// TwinCAT 3 PLC project AxisIaiLib
// Title: AxisIaiLibrary
// Company: Gema
// Author: RG
// ProjectVersion: 0.0.0.1
// ProgramVersion: 3.1.4024.0
// libraries:
//   Tc2_Standard, * (Beckhoff Automation GmbH)
//   TcoCore, 0.11.0.35 (Vortex.Library)
//   TcoData, 0.11.0.35 (Vortex.Library)
//   TcoDrivesBeckhoff, 0.11.0.35 (Vortex.Library)
//   TcoElements, 0.11.0.35 (Vortex.Library)
//   TcoIo, 0.11.0.35 (Vortex.Library)
//   TcoPneumatics, 0.11.0.35 (Vortex.Library)
//   TcoUtilities, 0.11.0.35 (Vortex.Library)
// project tree:
//   Context/ MainStation.TcPOU (not stored), PRG_TEST.TcPOU, TcUnitContext.TcPOU
//   IAI/Data types/ AxisLimits.TcDUT (not stored), IAIAxisStatus.TcDUT (not stored), IOAxis.TcDUT
//   IAI/Data types/Enum/ eSetPositionMode.TcDUT, E_AccelMode.TcDUT (not stored), E_RMod.TcDUT (not stored), E_StopMode.TcDUT (not stored)
//   IAI/Data types/Interfaces/ iSuperActuator.TcIO
//   IAI/Data types/In/Gateway/ GatewayStatus.TcDUT, StatusSignal0.TcDUT, StatusSignal1.TcDUT
//   IAI/Data types/In/ PlcIn.TcDUT, StatusIn.TcDUT
//   IAI/Data types/Out/ ControlOut.TcDUT, PlcOut.TcDUT
//   IAI/Data types/Out/Gateway/ ControlSignal0.TcDUT, ControlSignal1.TcDUT, GatewayControl.TcDUT (not stored)
//   IAI/Global Variables/ AxisStats.TcGVL, AxisStatsGlobal.TcGVL
//   IAI/IAI_Drive/TcoAxis/ AxisIAI.TcPOU, IAxisIAI.TcIO, Power.TcPOU
//   IAI/IAI_Drive/TcoAxis/AxisTasks/ ResetTask.TcPOU, SetPositionTask.TcPOU
//   IAI/IAI_Drive/TcoAxis/MotionTasks/ HaltTask.TcPOU, HomeTask.TcPOU, MoveAbsoluteTask.TcPOU, MoveRelativeTask.TcPOU, StopTask.TcPOU
// (motion and I/O tree: see PLC project axisiailibexample)
// real-time tasks:
//   TASK PlcTask: cycle T#10ms, priority 20, ADS port 350

// ---- IAI/Data types/Enum/eSetPositionMode.TcDUT
{attribute 'qualified_only'}
{attribute 'strict'}
TYPE
    eSetPositionMode :
    (
        Absolute := 0,
        Relative := 1
    );
END_TYPE

// ---- IAI/Data types/In/Gateway/GatewayStatus.TcDUT
TYPE
    GatewayStatus :
    STRUCT
        GatewayStatus0 : StatusSignal0;
        GatewayStatus1 : StatusSignal1;
        AnswerCmd      : WORD;
        Data0          : WORD;
        Data1          : WORD;
        Data2          : WORD;
        Data3          : WORD;
        UsedSpace      : WORD;
    END_STRUCT
END_TYPE

// ---- IAI/Data types/In/Gateway/StatusSignal0.TcDUT
TYPE
    StatusSignal0 :
    STRUCT
        //~
        ALMC1 : USINT; //Alarmcode from Gateway
        SEMG  : BIT;   //EMGIN off, --> Emergency Stop
        b9    : BIT;
        ALML  : BIT; // easy Error in Gateway, wrong Paramter
        ALMH  : BIT; // Sever Error in Gaateway, wrong Parameter, Rerstart req
        MODE  : BIT; // True if Mode = Manu
        ERRT  : BIT; //COMM Err between Axis and Gaetway
        LERC  : BIT; //ERror while Run  ERR-T or ERR-C in Gateway
        RUN   : BIT; //Running Gateway
    //~
    END_STRUCT
END_TYPE

// ---- IAI/Data types/In/Gateway/StatusSignal1.TcDUT
TYPE
    StatusSignal1 :
    STRUCT
        //~
        LNK0 : BIT; // zeigt aktive Achsennummer im Gateway
        LNK1 : BIT; // zeigt aktive Achsennummer im Gateway
        LNK2 : BIT; // zeigt aktive Achsennummer im Gateway
        LNK3 : BIT; // zeigt aktive Achsennummer im Gateway
        LNK4 : BIT; // zeigt aktive Achsennummer im Gateway
        LNK5 : BIT; // zeigt aktive Achsennummer im Gateway
        LNK6 : BIT; // zeigt aktive Achsennummer im Gateway
        LNK7 : BIT; // zeigt aktive Achsennummer im Gateway
        MNT0 : BIT; // Bit for Easy Error
        MNT1 : BIT; // Bit for Easy Error
        MNT2 : BIT; // Bit for Easy Error
        MNT3 : BIT; // Bit for Easy Error
        MNT4 : BIT; // Bit for Easy Error
        MNT5 : BIT; // Bit for Easy Error
        MNT6 : BIT; // Bit for Easy Error
        MNT7 : BIT; // Bit for Easy Error
    //~
    END_STRUCT
END_TYPE

// ---- IAI/Data types/In/PlcIn.TcDUT
TYPE
    PlcIn :
    //    (*PCON-CA output -> PLC input  - 32 bytes *)
    STRUCT
        CurrentPosition : DINT; (*Unit: 0,01mm*)
        CommandCurrent  : DINT; (*Unit: mA*)
        CurrentSpeed    : UINT; (*Unit: 0,01mm/s*)
        Unavailable1    : WORD; (*n+14;n+15*)
        AlarmCode       : UINT; (*0- no Error*)
        //        TotalMovingCount : UDINT; (*Unit: times*)
        //        TotalMovingDistance : UDINT; (*Unit: m*)
        StatusSignal : StatusIn;
    //        StatusSignal2 : WORD; (*n+30;n+31*)
    END_STRUCT
END_TYPE

// ---- IAI/Data types/In/StatusIn.TcDUT
TYPE
    StatusIn :
    STRUCT
        //~
        PEND  : BIT; //Signal wird true nach Abschluss Positionierung, on during Stop if Motor on
        HEND  : BIT; //True after Homeing, until Pos lost
        MOVE1 : BIT; //True while Moving
        ALM   : BIT; // true while Alarm
        SV    : BIT; //True when ready, (Servo On)
        PSFL  : BIT; //True while Error in SchubBetrieb
        bit6  : BIT;
        ALML  : BIT; //izi Error
        MEND  : BIT; //Signal True after Moving, Homing or Schubvorgang, False by Start new Movement
        bit9  : BIT;
        bit10 : BIT;
        bit11 : BIT;
        ZONE1 : BIT; // True when in Zone1
        ZONE2 : BIT;
        CRDY  : BIT; // Controller in Standby
        EMGS  : BIT; // Emergency Stop
    //~
    END_STRUCT
END_TYPE

// ---- IAI/Data types/IOAxis.TcDUT
TYPE
    IOAxis :
    STRUCT
        GateWayStatus  : GatewayStatus;
        GateWayControl : GatewayControl;
        PlcInFromAxis  : PlcIn;
        PlcOutToAxis   : PlcOut;
    END_STRUCT
END_TYPE

// ---- IAI/Data types/Out/ControlOut.TcDUT
TYPE
    ControlOut :
    STRUCT
        //~
        CSTR        : BIT; // Positionierungs Start, Trigger
        HOME        : BIT; // Referenzfahrt
        STP         : BIT; // PAuse
        RES         : BIT; // REset
        SON         : BIT; //Servo Ein
        JISL        : BIT; //Wechsel zwischen Jog/Inch Betrieb
        JVEL        : BIT; // Umschalten von Jog-Geschw/Schrittweite  S119 ANleitung
        JOGNegative : BIT; //-Jog
        JOGPositive : BIT; //+Jog
        b9          : BIT;
        b10         : BIT;
        b11         : BIT;
        PUSH        : BIT; //Schubbetrieb, True = Schubbetrieb, False = Positionierbetrieb
        DIR         : BIT; //Schubrichtung, True = Entgegen Refernezpunktrichtung
        INC         : BIT; //False= Absolute Positionsbefehle, True = Inkrementale
        BKRL        : BIT; //True = Bremsfreigabe, False = Bremse aktiv
    //~
    END_STRUCT
END_TYPE

// ---- IAI/Data types/Out/Gateway/ControlSignal0.TcDUT
TYPE
    ControlSignal0 :
    STRUCT
        //~
        b0  : BIT;
        b1  : BIT;
        b2  : BIT;
        b3  : BIT;
        b4  : BIT;
        b5  : BIT;
        b6  : BIT;
        b7  : BIT;
        b8  : BIT;
        b9  : BIT;
        b10 : BIT;
        b11 : BIT;
        b12 : BIT;
        RTE : BIT; //ERR-T oder ERR-C REset during Run
        b14 : BIT;
        MON : BIT; //must be on, Controll with Communication active
    //~
    END_STRUCT
END_TYPE

// ---- IAI/Data types/Out/Gateway/ControlSignal1.TcDUT
TYPE
    ControlSignal1 :
    STRUCT
        word1 : word;
    END_STRUCT
END_TYPE

// ---- IAI/Data types/Out/PlcOut.TcDUT
TYPE
    PlcOut :
    //    (*PCON-CA output -> PLC input  - 32 bytes *)
    STRUCT
        TargetPosition  : DINT := 1000; (*Unit: 0,01 mm*)
        PositioningBand : DINT := 10;   (*Unit: 0,01 mm or pressing width value*)
        Velocity        : UINT := 1;    (*Unit 0,01 mm/s*)
        //        ZoneBoundary_pos : DINT; (*Unit 0,01 mm*)
        //        ZoneBoundary_neg : DINT; (*Unit 0,01 mm*) (*pos >= neg!*)
        Accelerartion : UINT := 1; (*Acc und Dec Unit: 0,01 G*) (*Range 1.. 300*)
        //        Decelerartion : UINT; (*Unit: 0,01 G*) (*Range 1.. 300*)
        //        PressingCurrentLimitValue : UINT; (*Unit: %*) (*Range 0(0%) .. 510(200%)*)
        PushCurrentLimit : UINT := 1; (*Schubstrombegrenzung Unit: %*) (*Range 0(0%) .. 255(100%)*)
        ControlSignal    : ControlOut;                                 (*n+28;n+29*)
    //        ControlSignal2 : WORD; (*n+30;n+31*)
    END_STRUCT
END_TYPE

// ---- IAI/Global Variables/AxisStats.TcGVL
{attribute 'Tc2GvlVarNames'}
{attribute 'qualified_only'}
VAR_GLOBAL CONSTANT

    AxisLimitsRfid     : AxisLimits := (MaxAcceleration := 100, MaxPosition := 20000, MaxVelocity := 900);
    AxisLimitsAssembly : AxisLimits := (MaxAcceleration := 100, MaxPosition := 25000, MaxVelocity := 900);
    AxisLimitsMounting : AxisLimits := (MaxAcceleration := 100, MaxPosition := 40000, MaxVelocity := 840);

END_VAR

// ---- IAI/Global Variables/AxisStatsGlobal.TcGVL
{attribute 'Tc2GvlVarNames'}
{attribute 'qualified_only'}
VAR_GLOBAL CONSTANT
    MaxAcceleration1 : UINT := 100;
    MINPosition1     : DINT := 0;
    MaxPosition1     : DINT := 20000;
    MaxVelocity1     : UINT := 900;

    MaxAcceleration2 : UINT := 100;
    MINPosition2     : DINT := 0;
    MaxPosition2     : DINT := 25000;
    MaxVelocity2     : UINT := 900;

    MaxAcceleration3 : UINT := 100;
    MINPosition3     : DINT := 0;
    MaxPosition3     : DINT := 40000;
    MaxVelocity3     : UINT := 840;

END_VAR

// ---- IAI/Data types/Interfaces/iSuperActuator.TcIO
INTERFACE iSuperActuator

METHOD ErrorHandling : BOOL
VAR_INPUT
END_VAR
END_METHOD

PROPERTY IsError : bool
GET
END_GET
END_PROPERTY

METHOD ResetError : BOOL
VAR_INPUT
END_VAR
END_METHOD

END_INTERFACE

// ---- IAI/IAI_Drive/TcoAxis/IAxisIAI.TcIO
INTERFACE IAxisIAI

PROPERTY DriveRef : REFERENCE TO AxisIAI
GET
END_GET
END_PROPERTY

END_INTERFACE

// ---- Context/PRG_TEST.TcPOU
PROGRAM PRG_TEST
VAR
    _testSuite : TcUnitContext;
END_VAR

_testSuite.Run();
_testSuite.RtcSynchronize(true, '', 60);

END_PROGRAM

// ---- Context/TcUnitContext.TcPOU
FUNCTION_BLOCK TcUnitContext EXTENDS TcoCore.TcoContext
VAR
    _mainStation : MainStation(THIS^);

    {attribute addProperty Name "Versionsnummer Plc"}
    _sVersion : STRING(23);
    //~
    _stProgramVersion : ST_LibVersion;
    //~

END_VAR

(*~
    <docu>
        <summary>
            Main method of the TcoContext. This is the entry point of any control logic that belongs to this context.
            The call of this method is ensured by calling the <c>InstanceName.Run()</c> method, and it must not be called explicitly.
            This method is abstract, and it must be overridden in derived block.
        </summary>
    </docu>
~*)
METHOD PROTECTED Main

_mainStation();
END_METHOD

END_FUNCTION_BLOCK

// ---- IAI/IAI_Drive/TcoAxis/AxisIAI.TcPOU
FUNCTION_BLOCK AxisIAI EXTENDS TcoCore.TcoComponent IMPLEMENTS IAxisIAI, iSuperActuator
VAR_INPUT
    inEnabled : BOOL; // Power ein
END_VAR
VAR_OUTPUT
END_VAR
VAR_IN_OUT
    GateWayStatus  : GatewayStatus;
    GateWayControl : GatewayControl;

    DriveToPlc : PlcIn;
    PlcToDrive : PlcOut;

END_VAR
VAR
    //    _baseAxis : FB_SpecialControl(maxAcc := _maxAcc, minPos := _minPos, maxPos := _maxPos, maxVel := _maxVel);
    {attribute clr [ReadOnly()]}
    _axisStatus : IAIAxisStatus;
    _axisLimit  : AxisLimits;

    {attribute 'hide'}
    _sb        : TcoCore.StringBuilder;
    _errorDesc : string;
END_VAR
VAR
    _power : Power(THIS^);
    {attribute addProperty Name "Referenz (Aufpassen)"}
    _homeTask : HomeTask(THIS^);
    {attribute addProperty Name "<#Reset#>"}
    _resetTask : ResetTask(THIS^);
    {attribute addProperty Name "<#Set position#>"}
    _setPositionTask : SetPositionTask(THIS^);
    //	    {attribute addProperty Name "<#Jogging#>"}
    //    _jog : Jog(THIS^);
    {attribute addProperty Name "<#Stop#>"}
    _stopTask : StopTask(THIS^);
    {attribute addProperty Name "<#Halt#>"}
    _haltTask : HaltTask(THIS^);
    {attribute addProperty Name "<#Move relative#>"}
    _moveRelativeTask : MoveRelativeTask(THIS^);
    {attribute addProperty Name "<#Move absolute#>"}
    _moveAbsoluteTask : MoveAbsoluteTask(THIS^);
    //    {attribute addProperty Name "<#Move modulo#>"}
    //    _moveModuloTask : MoveModuloTask(THIS^);
    _faultTask : TcoCore.TcoTask(THIS^);
END_VAR


UpdateAxisStatus();

_power(inEnable := inEnabled);

_resetTask();

_homeTask();
_setPositionTask();
_stopTask();
_haltTask();
_moveRelativeTask();
_moveAbsoluteTask();
THIS^.Service();
//_moveModuloTask();

IF (_axisStatus.Error) THEN
    CASE _axisStatus.ErrorId OF
        111:
            _errorDesc := 'NotAus der Achse, bitte Checken';
        131:
            _errorDesc := 'Referenzfahrt nicht Complete';
        163:
            _errorDesc := 'Position Command Data invalid';
        193:
            _errorDesc := '0C1,Fehler Achse, Motorlast zu hoch aufgrund externer Kraft';
        333, 444, 555:
            _errorDesc := 'Servo ist aus';

    ELSE
        _errorDesc := 'For details see the service mode';

    END_CASE

    Messenger.Error
    (
        _sb.Clear()
            .Append('<#Drive error no #>')
            .Append(UDINT_TO_STRING(_axisStatus.ErrorId))
            .Append(': ')
            .Append(_errorDesc)
            .ToString()
    );

    _faultTask.ThrowWhen(TRUE);
END_IF;

UpdateAxisStatus();

PROPERTY AxisStatus : REFERENCE TO IAIAxisStatus
GET
UpdateAxisStatus();
AxisStatus REF= _axisStatus;
END_GET
END_PROPERTY

METHOD INTERNAL ClearError
_axisStatus.Error   := FALSE;
_axisStatus.ErrorId := 0;
END_METHOD

PROPERTY DriveRef : REFERENCE TO AxisIAI
GET
IF __ISVALIDREF(DriveRef) THEN
    DriveRef := THIS^;
end_if
END_GET
END_PROPERTY

METHOD ErrorHandling : BOOL
END_METHOD

PROPERTY FaultTask : TcoCore.ITcoTask
GET
FaultTask := _faultTask;
END_GET
END_PROPERTY

{attribute 'hide'}
METHOD FB_init : BOOL
VAR_INPUT
    bInitRetains : BOOL; // if TRUE, the retain variables are initialized (warm start / cold start)
    bInCopyCode  : BOOL; // if TRUE, the instance afterwards gets moved into the copy code (online change)
    ParentObject : ITcoObject;
    AxisLimits   : AxisLimits;
END_VAR
SUPER^.FB_init(bInitRetains, bInCopyCode, ParentObject);

THIS^._axisLimit := AxisLimits;
END_METHOD

METHOD Halt : ITcoTaskStatus
VAR_INPUT
    inDeceleration : UINT;
END_VAR
Halt := THIS^._haltTask.InvokeWithParams(inDeceleration := inDeceleration);
END_METHOD

PROPERTY HaltTask : TcoCore.ITcoTaskStatus
GET
HaltTask := _haltTask;
END_GET
END_PROPERTY

PROPERTY HomeTask : TcoCore.ITcoTaskStatus
GET
HomeTask := _homeTask;
END_GET
END_PROPERTY

PROPERTY isEnabled : BOOL
GET
isEnabled := inEnabled and DriveToPlc.StatusSignal.SV;
END_GET
END_PROPERTY

PROPERTY IsError : BOOL
GET
IsError := _faultTask.Error;
END_GET
END_PROPERTY

METHOD MoveAbsolute : ITcoTaskStatus
VAR_INPUT
    TargetPosition   : REAL;
    PositionBand     : REAL;
    Velocity         : UINT;
    Acceleration     : UINT;
    PushCurrentLimit : USINT;
END_VAR
MoveAbsolute := THIS^._moveAbsoluteTask.InvokeWithParams
(
    TargetPosition     := TargetPosition
    , PositionBand     := PositionBand
    , Velocity         := Velocity
    , Acceleration     := Acceleration
    , PushCurrentLimit := PushCurrentLimit
);
END_METHOD

PROPERTY MoveAbsoluteTask : TcoCore.ITcoTaskStatus
GET
MoveAbsoluteTask := _moveAbsoluteTask;
END_GET
END_PROPERTY

METHOD MoveHome : ITcoTaskStatus
VAR_INPUT
END_VAR
MoveHome := _homeTask.Invoke();
END_METHOD

METHOD MoveRelative : ITcoTaskStatus
VAR_INPUT
    Distance         : REAL;
    PositionBand     : REAL;
    Velocity         : UINT;
    Acceleration     : UINT;
    PushCurrentLimit : USINT;
END_VAR
MoveRelative := THIS^._moveRelativeTask.InvokeWithParams
(
    Distance           := Distance
    , Velocity         := Velocity
    , Acceleration     := Acceleration
    , PositionBand     := PositionBand
    , PushCurrentLimit := PushCurrentLimit
);
END_METHOD

PROPERTY MoveRelativeTask : TcoCore.ITcoTaskStatus
GET
MoveRelativeTask := _moveRelativeTask;
END_GET
END_PROPERTY

METHOD Reset : ITcoTaskStatus
Reset := THIS^._resetTask.Invoke();
ClearError();
END_METHOD

METHOD ResetError : BOOL
Restore();
END_METHOD

PROPERTY ResetTask : TcoCore.ITcoTaskStatus
GET
ResetTask := _resetTask;
END_GET
END_PROPERTY

(*~
    <docu>
        <summary>
            Restores this instance to the Ready state. Can be called explicitly or from within one of the restore mechanisms.
        </summary>
    </docu>
~*)
METHOD Restore : ITcoRestorable
Reset();
RestoreTasks();
END_METHOD

METHOD RestoreTasks : ITcoRestorable
VAR_INPUT
END_VAR
//Restore all
_homeTask.Restore();
_resetTask.Restore();
_setPositionTask.Restore();
_stopTask.Restore();
_haltTask.Restore();
_moveRelativeTask.Restore();
_moveAbsoluteTask.Restore();
_resetTask.Restore();
_faultTask.Restore();
END_METHOD

(*~
    <docu>
        <summary>
            Custom service (manual, maintenance) logic.
            This method must be implemented in derived class.
        </summary>
    </docu>
~*)
METHOD PROTECTED ServiceMode
//_jog.Service();
END_METHOD

METHOD INTERNAL SetErrorID
VAR_INPUT
    inErrorId : UDINT;
END_VAR
_axisStatus.Error := TRUE;

IF inErrorId <> 0 THEN
    _axisStatus.ErrorId := inErrorId;
ELSIF DriveToPlc.StatusSignal.EMGS THEN
    _axisStatus.ErrorId := 111;
END_IF
END_METHOD

METHOD SetPosition : ITcoTaskStatus
VAR_INPUT
    inPosition : LREAL;
    inMode     : eSetPositionMode;
END_VAR
SetPosition := THIS^._setPositionTask.InvokeWithParams(inPosition := inPosition, inMode := inMode);
END_METHOD

PROPERTY SetPositionTask : TcoCore.ITcoTaskStatus
GET
SetPositionTask := _setPositionTask;
END_GET
END_PROPERTY

METHOD Stop : ITcoTaskStatus
VAR_INPUT
    inDeceleration : UINT;
END_VAR
Stop := THIS^._stopTask.InvokeWithParams(inDeceleration := inDeceleration);
END_METHOD

PROPERTY StopTask : TcoCore.ITcoTaskStatus
GET
StopTask := _stopTask;
END_GET
END_PROPERTY

METHOD INTERNAL UpdateAxisStatus
VAR
    _message : STRING(125);
END_VAR
_axisStatus.ActPos := DriveToPLC.CurrentPosition / 100.0;
//_axisStatus.ModuloActPos := AxisRef.NcToPlc.ModuloActPos;
//_axisStatus.ModuloActTurns := AxisRef.NcToPlc.ModuloActTurns;
_axisStatus.ActVelo := DriveToPLC.CurrentSpeed;
//_axisStatus.ActAcc := AxisRef.NcToPlc.ActAcc;
_axisStatus.ActTorque := DriveToPLC.CommandCurrent;
//_axisStatus.CmdNo := AxisRef.NcToPlc.CmdNo;
//_axisStatus.CmdState := AxisRef.NcToPlc.CmdState;

//IF NOT Tc2MC2_TO_Tco_AxisStates(AxisRef.Status.MotionState, _axisStatus.MotionState) THEN
//    _message := Tc2_Standard
//        .CONCAT('Unable to cast AxisRef.Status.MotionState variable of type Tc2_MC2.MC_AxisStates (', TO_STRING(AxisRef.Status.MotionState));

//    _message := Tc2_Standard.CONCAT(_message, ') to the type TcoDrivesBeckhoff.eAxisStates!!!');
//    THIS^.Messenger.Post(_message, TcoCore.eMessageCategory.ProgrammingError);
//END_IF

//AlarmCodes ausprogrammieren (alle Gateway ALarmcodes etc.)
IF (DriveToPLC.StatusSignal.ALM OR DriveToPLC.StatusSignal.ALML or DriveToPlc.StatusSignal.EMGS) THEN
    SetErrorID(DriveToPlc.AlarmCode);
END_IF

//_axisStatus.ErrorStop := AxisRef.Status.ErrorStop;
//_axisStatus.Disabled := AxisRef.Status.Disabled;
//_axisStatus.Stopping := AxisRef.Status.Stopping;
_axisStatus.StandStill       := NOT DriveToPLC.StatusSignal.MOVE1;
_axisStatus.DiscreteMotion   := PLCToDrive.ControlSignal.JISL;
_axisStatus.ContinuousMotion := NOT PLCToDrive.ControlSignal.JISL;
_axisStatus.AbsoluteMotion   := NOT PLCToDrive.ControlSignal.INC;
_axisStatus.RelativeMotion   := PLCToDrive.ControlSignal.INC;
//_axisStatus.SynchronizedMotion := AxisRef.Status.SynchronizedMotion;
_axisStatus.Homing := DriveToPLC.StatusSignal.MOVE1 AND NOT DriveToPLC.StatusSignal.HEND;
//_axisStatus.ConstantVelocity := AxisRef.Status.ConstantVelocity;
//_axisStatus.Accelerating := AxisRef.Status.Accelerating;
//_axisStatus.Decelerating := AxisRef.Status.Decelerating;
_axisStatus.Operational := GateWayStatus.GatewayStatus0.RUN;
//_axisStatus.ControlLoopClosed := AxisRef.Status.ControlLoopClosed;
//_axisStatus.HasJob := AxisRef.Status.HasJob;
_axisStatus.HasBeenStopped := PLCToDrive.ControlSignal.STP;
//_axisStatus.NewTargetPosition := AxisRef.Status.NewTargetPosition;
_axisStatus.InPositionArea    := DriveToPLC.StatusSignal.PEND and not DriveToPlc.StatusSignal.MOVE1;
_axisStatus.InTargetPosition1 := DriveToPLC.StatusSignal.ZONE1;
_axisStatus.InTargetPosition2 := DriveToPLC.StatusSignal.ZONE2;
_axisStatus.Homed             := DriveToPLC.StatusSignal.HEND;
//_axisStatus.HomingBusy := AxisRef.Status.HomingBusy;
//_axisStatus.MotionCommandsLocked := AxisRef.Status.MotionCommandsLocked;
//_axisStatus.SoftLimitMinExceeded := AxisRef.Status.SoftLimitMinExceeded;
//_axisStatus.SoftLimitMaxExceeded := AxisRef.Status.SoftLimitMaxExceeded;
_axisStatus.Moving            := DriveToPLC.StatusSignal.MOVE1;
_axisStatus.PositiveDirection := PLCToDrive.ControlSignal.DIR;
_axisStatus.NegativeDirection := NOT PLCToDrive.ControlSignal.DIR;
_axisStatus.NotMoving         := NOT DriveToPLC.StatusSignal.MOVE1;
//_axisStatus.Compensating := AxisRef.Status.Compensating;
//_axisStatus.ExtSetPointGenEnabled := AxisRef.Status.ExtSetPointGenEnabled;
//_axisStatus.ExternalLatchValid := AxisRef.Status.ExternalLatchValid;
//_axisStatus.CamDataQueued := AxisRef.Status.CamDataQueued;
//_axisStatus.CamTableQueued := AxisRef.Status.CamTableQueued;
//_axisStatus.CamScalingPending := AxisRef.Status.CamScalingPending;
//_axisStatus.CmdBuffered := AxisRef.Status.CmdBuffered;
//_axisStatus.PTPmode := AxisRef.Status.PTPmode;
_axisStatus.DriveDeviceError :=
    GateWayStatus.GatewayStatus0.ALMH OR GateWayStatus.GatewayStatus0.ALML OR GateWayStatus.GatewayStatus0.LERC;

_axisStatus.IoDataInvalid := GateWayStatus.GatewayStatus0.ERRT;
_axisStatus.Coupled1      := GateWayStatus.GatewayStatus1.LNK0;
_axisStatus.Coupled2      := GateWayStatus.GatewayStatus1.LNK2;
_axisStatus.Coupled3      := GateWayStatus.GatewayStatus1.LNK4;
_axisStatus.Coupled4      := GateWayStatus.GatewayStatus1.LNK6;

//_axisStatus.OpMode.PositionAreaMonitoring := AxisRef.Status.OpMode.PositionAreaMonitoring;
//_axisStatus.OpMode.TargetPositionMonitoring := AxisRef.Status.OpMode.TargetPositionMonitoring;
//_axisStatus.OpMode.LoopMode := AxisRef.Status.OpMode.LoopMode;
//_axisStatus.OpMode.MotionMonitoring := AxisRef.Status.OpMode.MotionMonitoring;
//_axisStatus.OpMode.PEHTimeMonitoring := AxisRef.Status.OpMode.PEHTimeMonitoring;
//_axisStatus.OpMode.BacklashCompensation := AxisRef.Status.OpMode.BacklashCompensation;
//_axisStatus.OpMode.Modulo := AxisRef.Status.OpMode.Modulo;
//_axisStatus.OpMode.PositionLagMonitoring := AxisRef.Status.OpMode.PositionLagMonitoring;
//_axisStatus.OpMode.VelocityLagMonitoring := AxisRef.Status.OpMode.VelocityLagMonitoring;
//_axisStatus.OpMode.SoftLimitMinMonitoring := AxisRef.Status.OpMode.SoftLimitMinMonitoring;
//_axisStatus.OpMode.SoftLimitMaxMonitoring := AxisRef.Status.OpMode.SoftLimitMaxMonitoring;
//_axisStatus.OpMode.PositionCorrection := AxisRef.Status.OpMode.PositionCorrection;
END_METHOD

END_FUNCTION_BLOCK

// ---- IAI/IAI_Drive/TcoAxis/Power.TcPOU
FUNCTION_BLOCK Power EXTENDS TcoCore.TcoObject IMPLEMENTS IAxisIAI
VAR_INPUT
    inEnable : BOOL;
    //    inEnablePositive : BOOL;
    //    inEnableNegative : BOOL;
    //    inOverride : LREAL;
    //	inIsServiceMode : BOOL;
END_VAR
VAR
    {attribute addProperty Name "<#Power enable#>"}
    {attribute addProperty StateOnDesc "<#Enabled#>"}
    {attribute addProperty StateOffDesc "<#Disabled#>"}
    _driveEnableLocalTask : TcoCore.TcoToggleTask(THIS^, FALSE);
    //    {attribute addProperty Name "<#Enable positive#>"}
    //	{attribute addProperty StateOnDesc "<#Enabled#>"}
    //	{attribute addProperty StateOffDesc "<#Disabled#>"}
    //    _driveEnablePositiveLocalTask : TcoCore.TcoToggleTask(THIS^,FALSE);
    //    {attribute addProperty Name "<#Enable negative#>"}
    //	{attribute addProperty StateOnDesc "<#Enabled#>"}
    //	{attribute addProperty StateOffDesc "<#Disabled#>"}
    //    _driveEnableNegativeLocalTask : TcoCore.TcoToggleTask(THIS^,FALSE);
END_VAR


_driveEnableLocalTask.Run();
//_driveEnablePositiveLocalTask.Run();
//_driveEnableNegativeLocalTask.Run();

IF inEnable THEN
    _driveEnableLocalTask.On();
ELSE
    _driveEnableLocalTask.Off();
END_IF

DriveRef.PlcToDrive.ControlSignal.SON := _driveEnableLocalTask.IsOn;

PROPERTY DriveRef : REFERENCE TO AxisIAI
GET
VAR
    _drive : POINTER TO AxisIAI;
END_VAR
IF __QUERYPOINTER(THIS^._ParentObject, _drive) THEN
    DriveRef REF= _drive^;
END_IF
END_GET
END_PROPERTY

METHOD FB_init : BOOL
VAR_INPUT
    bInitRetains : BOOL; // if TRUE, the retain variables are initialized (warm start / cold start)
    bInCopyCode  : BOOL; // if TRUE, the instance afterwards gets moved into the copy code (online change)
    ParentObject : TcoCore.ITcoObject;
END_VAR
SUPER^.FB_init(bInitRetains := bInitRetains, bInCopyCode := bInCopyCode, ParentObject := ParentObject);
END_METHOD

END_FUNCTION_BLOCK

// ---- IAI/IAI_Drive/TcoAxis/MotionTasks/HomeTask.TcPOU
FUNCTION_BLOCK HomeTask EXTENDS TcoCore.TcoTask IMPLEMENTS IAxisIAI
VAR
    {attribute 'hide'}
    _message : STRING(125);

    HomeTrig : R_TRIG;
    _error   : bool;
END_VAR

THIS^.Enabled :=
    NOT DriveRef.HaltTask.Busy AND NOT DriveRef.MoveAbsoluteTask.Busy AND NOT DriveRef.MoveRelativeTask.Busy;

IF (THIS^.Execute()) THEN
    DriveRef.PlcToDrive.ControlSignal.HOME := TRUE;
    HomeTrig(CLK := DriveRef.AxisStatus.Homed);

    THIS^.DoneWhen(HomeTrig.Q);

    IF DriveRef.AxisStatus.Error THEN
        _error := true;
    END_IF

    THIS^.ThrowWhen(DriveRef.AxisStatus.Error or not DriveRef.PlcToDrive.ControlSignal.SON);
    THIS^.Messenger.Error('Axis Error while Homing').Pin();
END_IF

PROPERTY DriveRef : REFERENCE TO AxisIAI
GET
VAR
    _drive : POINTER TO AxisIAI;
END_VAR
IF __QUERYPOINTER(THIS^._ParentObject, _drive) THEN
    DriveRef REF= _drive^;
END_IF
END_GET
END_PROPERTY

{attribute 'hide'}
METHOD PUBLIC FB_init : BOOL
VAR_INPUT
    bInitRetains : BOOL; // if TRUE, the retain variables are initialized (warm start / cold start)
    bInCopyCode  : BOOL; // if TRUE, the instance afterwards gets moved into the copy code (online change)
    ParentObject : ITcoObject;
END_VAR
SUPER^.FB_init(bInitRetains := bInitRetains, bInCopyCode := bInCopyCode, ParentObject := ParentObject);
END_METHOD

(*~
    <docu>
        <summary>
            Executes when task reaches the ```Done``` state .
        </summary>
    </docu>
~*)
METHOD PROTECTED OnDone
DriveRef.PlcToDrive.ControlSignal.HOME := FALSE;
DriveRef.Restore();
END_METHOD

(*~
    <docu>
        <summary>
            Executes when task reaches the ```Error``` state.
            <para>
                Do not confuse with <see cref="PlcDocu.TcoCore.TcoTask.WhileError()"/>, that is called cyclically until '''Error''' state is left.
            </para>
        </summary>
    </docu>
~*)
METHOD PROTECTED OnError
DriveRef.SetErrorID(333);
END_METHOD

(*~
    <docu>
        <summary>
            Restores this instance to the Ready state. Can be called explicitly or from within one of the restore mechanisms.
            <para>
                See also <see cref="PlcDocu.TcoCore.TcoTask.AutoRestorable()"/>
            </para>
        </summary>
    </docu>
~*)
METHOD Restore : ITcoRestorable
DriveRef.PlcToDrive.ControlSignal.HOME := FALSE;
Super^.Restore();
END_METHOD

END_FUNCTION_BLOCK

// ---- IAI/IAI_Drive/TcoAxis/MotionTasks/HaltTask.TcPOU
FUNCTION_BLOCK HaltTask EXTENDS TcoCore.TcoTask IMPLEMENTS IAxisIAI
VAR
    {attribute addProperty Name "<#Deceleration#>"}
    _deceleration : UINT;
END_VAR


IF Execute() THEN
    DriveRef.PlcToDrive.ControlSignal.STP := TRUE;

    DoneWhen(DriveRef.AxisStatus.NotMoving);
    ThrowWhen(DriveRef.AxisStatus.Error);
END_IF

PROPERTY DriveRef : REFERENCE TO AxisIAI
GET
VAR
    _drive : POINTER TO AxisIAI;
END_VAR
IF __QUERYPOINTER(THIS^._ParentObject, _drive) THEN
    DriveRef REF= _drive^;
END_IF
END_GET
END_PROPERTY

METHOD PUBLIC FB_init : BOOL
VAR_INPUT
    bInitRetains : BOOL; // if TRUE, the retain variables are initialized (warm start / cold start)
    bInCopyCode  : BOOL; // if TRUE, the instance afterwards gets moved into the copy code (online change)
    ParentObject : ITcoObject;
END_VAR
SUPER^.FB_init(bInitRetains := bInitRetains, bInCopyCode := bInCopyCode, ParentObject := ParentObject);
END_METHOD

METHOD INTERNAL InvokeWithParams : ITcoTaskStatus
VAR_INPUT
    inDeceleration : UINT;
END_VAR
_deceleration    := inDeceleration;
InvokeWithParams := THIS^.Invoke();
END_METHOD

(*~
    <docu>
        <summary>
            Executes when task reaches the ```Done``` state .
        </summary>
    </docu>
~*)
METHOD PROTECTED OnDone
Restore();
DriveRef.Restore();
END_METHOD

(*~
    <docu>
        <summary>
            Restores this instance to the Ready state. Can be called explicitly or from within one of the restore mechanisms.
            <para>
                See also <see cref="PlcDocu.TcoCore.TcoTask.AutoRestorable()"/>
            </para>
        </summary>
    </docu>
~*)
METHOD Restore : ITcoRestorable
SUPER^.Restore();
END_METHOD

END_FUNCTION_BLOCK

// ---- IAI/IAI_Drive/TcoAxis/MotionTasks/MoveAbsoluteTask.TcPOU
FUNCTION_BLOCK MoveAbsoluteTask EXTENDS TcoCore.TcoTask IMPLEMENTS IAxisIAI
VAR
    {attribute addProperty Maximum 11.0f}
    {attribute addProperty Name "<#Position in mm#>"}
    {attribute addProperty Units "mm"}
    _position : REAL := 10.0;
    {attribute addProperty Name "<#Positionierbereich in mm#>"}
    _positionBand : REAL := 0.1;
    {attribute addProperty Name "<#Geschwindigkeit in mm/s#>"}
    _velocity : UINT := 10;
    {attribute addProperty Name "<#Beschleunigung (0 - 100)#>"}
    _acceleration : UINT := 10;
    {attribute addProperty Name "<#Schubstrombegrenzung#>"}
    _pushCurrentLimit : USINT := 10;
    _doneTrig         : R_TRIG;
    _moveTrig         : TC2_Standard.R_TRIG;
    //~
    _state :
        (Init
        , Moving
        , Stopping);
    //~
    _startCount : ULINT;
END_VAR

THIS^.Enabled := NOT DriveRef.HaltTask.Busy AND NOT DriveRef.MoveRelativeTask.Busy AND NOT DriveRef.HomeTask.Busy;
_doneTrig();

IF Execute() THEN
    DriveRef.PlcToDrive.ControlSignal.INC := FALSE;
    DriveRef.PlcToDrive.Accelerartion     := _acceleration;
    DriveRef.PlcToDrive.PushCurrentLimit  := _pushCurrentLimit;
    //for Visu
    DriveRef.PlcToDrive.PositioningBand    := REAL_TO_DINT((_positionBand * 100));
    DriveRef.PlcToDrive.TargetPosition     := REAL_TO_DINT((_position * 100));
    DriveRef.PlcToDrive.Velocity           := _velocity;
    DriveRef.PlcToDrive.ControlSignal.CSTR := TRUE;

    IF THIS^.ElapsedTime >= T#20MS THEN
        DoneWhen(DriveRef.AxisStatus.NotMoving);
        DriveRef.PlcToDrive.ControlSignal.CSTR := FALSE;

        IF DriveRef.DriveToPlc.CurrentPosition = REAL_TO_DINT((_position * 100)) THEN
            DoneWhen(TRUE);
            DriveRef.PlcToDrive.ControlSignal.CSTR := FALSE;
        END_IF
    END_IF

    ThrowWhen(DriveRef.AxisStatus.Error);
END_IF

PROPERTY DriveRef : REFERENCE TO AxisIAI
GET
VAR
    _drive : POINTER TO AxisIAI;
END_VAR
IF __QUERYPOINTER(THIS^._ParentObject, _drive) THEN
    DriveRef REF= _drive^;
END_IF
END_GET
END_PROPERTY

METHOD PUBLIC FB_init : BOOL
VAR_INPUT
    bInitRetains : BOOL; // if TRUE, the retain variables are initialized (warm start / cold start)
    bInCopyCode  : BOOL; // if TRUE, the instance afterwards gets moved into the copy code (online change)
    ParentObject : ITcoObject;
END_VAR
SUPER^.FB_init(bInitRetains := bInitRetains, bInCopyCode := bInCopyCode, ParentObject := ParentObject);
END_METHOD

METHOD INTERNAL InvokeWithParams : ITcoTaskStatus
VAR_INPUT
    TargetPosition   : REAL;
    PositionBand     : REAL;
    Velocity         : UINT;
    Acceleration     : UINT;
    PushCurrentLimit : USINT;
END_VAR
_position         := TargetPosition;
_positionBand     := PositionBand;
_velocity         := Velocity;
_acceleration     := Acceleration;
_pushCurrentLimit := PushCurrentLimit;
InvokeWithParams  := THIS^.Invoke();
END_METHOD

(*~
    <docu>
        <summary>
            Executes when task is aborted.
        </summary>
    </docu>
~*)
METHOD PROTECTED OnAbort

THIS^.DriveRef.AxisStatus.HasBeenStopped    := TRUE;
THIS^.DriveRef.PlcToDrive.ControlSignal.RES := TRUE;
_state                                      := Init;
DriveRef.PlcToDrive.ControlSignal.CSTR      := FALSE;
//_mcMoveAbsolute(Axis := _axisRef, Execute := FALSE);
END_METHOD

(*~
    <docu>
        <summary>
            Executes when task reaches the ```Done``` state .
        </summary>
    </docu>
~*)
METHOD PROTECTED OnDone
DriveRef.PlcToDrive.ControlSignal.CSTR := FALSE;
_state                                 := Init;
//THIS^.Restore();
END_METHOD

(*~
    <docu>
        <summary>
            Executes when task reaches the ```Error``` state.
            <para>
                Do not confuse with <see cref="PlcDocu.TcoCore.TcoTask.WhileError()"/>, that is called cyclically until '''Error''' state is left.
            </para>
        </summary>
    </docu>
~*)
METHOD PROTECTED OnError
DriveRef.PlcToDrive.ControlSignal.CSTR := FALSE;
DriveRef.SetErrorID(DriveRef.AxisStatus.ErrorId);
END_METHOD

(*~
    <docu>
        <summary>
            Restores this instance to the Ready state. Can be called explicitly or from within one of the restore mechanisms.
            <para>
                See also <see cref="PlcDocu.TcoCore.TcoTask.AutoRestorable()"/>
            </para>
        </summary>
    </docu>
~*)
METHOD Restore : ITcoRestorable

DriveRef.PlcToDrive.ControlSignal.CSTR := FALSE;
DriveRef.PlcToDrive.ControlSignal.STP  := FALSE;
_state                                 := Init;
SUPER^.Restore();
END_METHOD

END_FUNCTION_BLOCK

// ---- IAI/IAI_Drive/TcoAxis/MotionTasks/MoveRelativeTask.TcPOU
FUNCTION_BLOCK MoveRelativeTask EXTENDS TcoCore.TcoTask IMPLEMENTS IAxisIAI
VAR
    {attribute addProperty Name "<#Distance#>"}
    _distance : REAL;
    {attribute addProperty Name "<#Positionierbereich in mm#>"}
    _positionBand : REAL := 0.1;
    {attribute addProperty Name "<#Geschwindigkeit in mm/s#>"}
    _velocity : UINT := 10;
    {attribute addProperty Name "<#Beschleunigung (0 - 100)#>"}
    _acceleration : UINT := 10;
    {attribute addProperty Name "<#Schubstrombegrenzung#>"}
    _pushCurrentLimit : USINT := 10;
    _doneTrig         : R_TRIG;
    _move             : BOOL := TRUE;
    _targetDest       : REAL;
    _actPos           : REAL;
    _executeTr        : R_TRIG;
END_VAR

THIS^.Enabled := NOT DriveRef.HaltTask.Busy AND NOT DriveRef.MoveAbsoluteTask.Busy AND NOT DriveRef.HomeTask.Busy;

_executeTr(CLK := Execute());

IF Execute() THEN
    DriveRef.PlcToDrive.ControlSignal.INC := TRUE;
    DriveRef.PlcToDrive.Accelerartion     := _acceleration;
    //for Visu
    DriveRef.PlcToDrive.PositioningBand := REAL_TO_DINT((_positionBand * 100));
    DriveRef.PlcToDrive.TargetPosition  := REAL_TO_DINT((_distance * 100));

    IF _executeTr.Q THEN
        _targetDest                            := DriveRef.AxisStatus.ActPos + _distance;
        DriveRef.PlcToDrive.ControlSignal.CSTR := TRUE;
    END_IF

    DriveRef.PlcToDrive.Velocity := _velocity;
    _actPos                      := DriveRef.AxisStatus.ActPos;

    IF THIS^.ElapsedTime >= T#20MS THEN
        IF (ABS(_targetDest - DriveRef.AxisStatus.ActPos) <= _positionBand) THEN
            DoneWhen(TRUE);
            DriveRef.PlcToDrive.ControlSignal.CSTR := FALSE;
        END_IF
    END_IF

    ThrowWhen(driveRef.AxisStatus.Error);
END_IF

PROPERTY DriveRef : REFERENCE TO AxisIAI
GET
VAR
    _drive : POINTER TO AxisIAI;
END_VAR
IF __QUERYPOINTER(THIS^._ParentObject, _drive) THEN
    DriveRef REF= _drive^;
END_IF
END_GET
END_PROPERTY

METHOD PUBLIC FB_init : BOOL
VAR_INPUT
    bInitRetains : BOOL; // if TRUE, the retain variables are initialized (warm start / cold start)
    bInCopyCode  : BOOL; // if TRUE, the instance afterwards gets moved into the copy code (online change)
    ParentObject : ITcoObject;
END_VAR
SUPER^.FB_init(bInitRetains := bInitRetains, bInCopyCode := bInCopyCode, ParentObject := ParentObject);
END_METHOD

METHOD INTERNAL InvokeWithParams : ITcoTaskStatus
VAR_INPUT
    Distance         : REAL;
    PositionBand     : REAL;
    Velocity         : UINT;
    Acceleration     : UINT;
    PushCurrentLimit : USINT;
END_VAR
_distance         := Distance;
_positionBand     := PositionBand;
_velocity         := Velocity;
_acceleration     := Acceleration;
_pushCurrentLimit := PushCurrentLimit;
InvokeWithParams  := THIS^.Invoke();
END_METHOD

(*~
    <docu>
        <summary>
            Executes when task is aborted.
        </summary>
    </docu>
~*)
METHOD PROTECTED OnAbort
DriveRef.PlcToDrive.ControlSignal.CSTR      := FALSE;
THIS^.DriveRef.AxisStatus.HasBeenStopped    := TRUE;
THIS^.DriveRef.PlcToDrive.ControlSignal.RES := TRUE;

//SUPER^.Restore();
//_mcMoveAbsolute(Axis := _axisRef, Execute := FALSE);
END_METHOD

(*~
    <docu>
        <summary>
            Executes when task reaches the ```Done``` state .
        </summary>
    </docu>
~*)
METHOD PROTECTED OnDone
//DriveRef.PlcToDrive.ControlSignal.CSTR := FALSE;
//DriveRef.Restore();
END_METHOD

(*~
    <docu>
        <summary>
            Executes when task reaches the ```Error``` state.
            <para>
                Do not confuse with <see cref="PlcDocu.TcoCore.TcoTask.WhileError()"/>, that is called cyclically until '''Error''' state is left.
            </para>
        </summary>
    </docu>
~*)
METHOD PROTECTED OnError
DriveRef.PlcToDrive.ControlSignal.CSTR := FALSE;
DriveRef.SetErrorID(DriveRef.AxisStatus.ErrorId);
END_METHOD

(*~
    <docu>
        <summary>
            Restores this instance to the Ready state. Can be called explicitly or from within one of the restore mechanisms.
            <para>
                See also <see cref="PlcDocu.TcoCore.TcoTask.AutoRestorable()"/>
            </para>
        </summary>
    </docu>
~*)
METHOD Restore : ITcoRestorable
DriveRef.PlcToDrive.ControlSignal.STP  := FALSE;
DriveRef.PlcToDrive.ControlSignal.CSTR := FALSE;
SUPER^.Restore();
END_METHOD

END_FUNCTION_BLOCK

// ---- IAI/IAI_Drive/TcoAxis/AxisTasks/ResetTask.TcPOU
FUNCTION_BLOCK ResetTask EXTENDS TcoCore.TcoTask IMPLEMENTS IAxisIAI
VAR

END_VAR

THIS^.Enabled := NOT DriveRef.AxisStatus.Moving;

IF Execute() THEN
    DriveRef.FaultTask.Restore();

    IF DriveRef.PlcToDrive.ControlSignal.RES THEN
        DriveRef.PlcToDrive.ControlSignal.RES := FALSE;
    ELSE
        DriveRef.PlcToDrive.ControlSignal.RES := TRUE;
        DriveRef.ClearError();

    END_IF

    DriveRef.PlcToDrive.ControlSignal.INC := FALSE;
    DriveRef.PlcToDrive.Accelerartion     := 1;
    DriveRef.PlcToDrive.PushCurrentLimit  := 1;
    DriveRef.PlcToDrive.PositioningBand   := 1;
    DriveRef.PlcToDrive.TargetPosition    := 1;
    DriveRef.PlcToDrive.Velocity          := 1;

    DoneWhen(NOT (DriveRef.DriveToPlc.StatusSignal.ALM OR DriveRef.AxisStatus.Error));
END_IF

PROPERTY DriveRef : REFERENCE TO AxisIAI
GET
VAR
    _drive : POINTER TO AxisIAI;
END_VAR
IF __QUERYPOINTER(THIS^._ParentObject, _drive) THEN
    DriveRef REF= _drive^;
END_IF
END_GET
END_PROPERTY

METHOD PUBLIC FB_init : BOOL
VAR_INPUT
    bInitRetains : BOOL; // if TRUE, the retain variables are initialized (warm start / cold start)
    bInCopyCode  : BOOL; // if TRUE, the instance afterwards gets moved into the copy code (online change)
    ParentObject : ITcoObject;
END_VAR
SUPER^.FB_init(bInitRetains := bInitRetains, bInCopyCode := bInCopyCode, ParentObject := ParentObject);
END_METHOD

(*~
    <docu>
        <summary>
            Executes when task reaches the ```Done``` state .
        </summary>
    </docu>
~*)
METHOD PROTECTED OnDone
DriveRef.RestoreTasks();
Restore();
DriveRef.ClearError();

DriveRef.PlcToDrive.ControlSignal.RES := FALSE;
END_METHOD

(*~
    <docu>
        <summary>
            Restores this instance to the Ready state. Can be called explicitly or from within one of the restore mechanisms.
            <para>
                See also <see cref="PlcDocu.TcoCore.TcoTask.AutoRestorable()"/>
            </para>
        </summary>
    </docu>
~*)
METHOD Restore : ITcoRestorable
SUPER^.Restore();
END_METHOD

END_FUNCTION_BLOCK

// ---- IAI/IAI_Drive/TcoAxis/AxisTasks/SetPositionTask.TcPOU
FUNCTION_BLOCK SetPositionTask EXTENDS TcoCore.TcoTask IMPLEMENTS IAxisIAI
VAR
    {attribute addProperty Name "<#Position#>"}
    _position : LREAL;
    {attribute addProperty Name "<#Mode#>"}
    _mode : eSetPositionMode;
END_VAR
VAR
    {attribute 'hide'}
    _message : STRING(125);
END_VAR


IF Execute() THEN
    //   DriveRef.AxisStatus.OpMode
    DoneWhen(TRUE);
    //    ThrowWhen(_mcSetPosition.Error);
END_IF

PROPERTY DriveRef : REFERENCE TO AxisIAI
GET
VAR
    _drive : POINTER TO AxisIAI;
END_VAR
IF __QUERYPOINTER(THIS^._ParentObject, _drive) THEN
    DriveRef REF= _drive^;
END_IF
END_GET
END_PROPERTY

METHOD PUBLIC FB_init : BOOL
VAR_INPUT
    bInitRetains : BOOL; // if TRUE, the retain variables are initialized (warm start / cold start)
    bInCopyCode  : BOOL; // if TRUE, the instance afterwards gets moved into the copy code (online change)
    ParentObject : ITcoObject;
END_VAR
SUPER^.FB_init(bInitRetains := bInitRetains, bInCopyCode := bInCopyCode, ParentObject := ParentObject);
END_METHOD

METHOD INTERNAL InvokeWithParams : ITcoTaskStatus
VAR_INPUT
    inPosition : LREAL;
    inMode     : eSetPositionMode;
END_VAR
_position        := inPosition;
_mode            := inMode;
InvokeWithParams := THIS^.Invoke();
END_METHOD

(*~
    <docu>
        <summary>
            Restores this instance to the Ready state. Can be called explicitly or from within one of the restore mechanisms.
            <para>
                See also <see cref="PlcDocu.TcoCore.TcoTask.AutoRestorable()"/>
            </para>
        </summary>
    </docu>
~*)
METHOD Restore : ITcoRestorable
SUPER^.Restore();
END_METHOD

END_FUNCTION_BLOCK

// ---- IAI/IAI_Drive/TcoAxis/MotionTasks/StopTask.TcPOU
FUNCTION_BLOCK StopTask EXTENDS TcoCore.TcoTask IMPLEMENTS IAxisIAI
VAR
    {attribute addProperty Name "<#Deceleration#>"}
    _deceleration : UINT;
END_VAR


IF Execute() THEN
    DriveRef.PlcToDrive.ControlSignal.STP := TRUE;
    DriveRef.PlcToDrive.ControlSignal.RES := TRUE;

    DoneWhen(DriveRef.AxisStatus.NotMoving);
    ThrowWhen(DriveRef.AxisStatus.Error);
END_IF

PROPERTY DriveRef : REFERENCE TO AxisIAI
GET
VAR
    _drive : POINTER TO AxisIAI;
END_VAR
IF __QUERYPOINTER(THIS^._ParentObject, _drive) THEN
    DriveRef REF= _drive^;
END_IF
END_GET
END_PROPERTY

METHOD PUBLIC FB_init : BOOL
VAR_INPUT
    bInitRetains : BOOL; // if TRUE, the retain variables are initialized (warm start / cold start)
    bInCopyCode  : BOOL; // if TRUE, the instance afterwards gets moved into the copy code (online change)
    ParentObject : ITcoObject;
END_VAR
SUPER^.FB_init(bInitRetains := bInitRetains, bInCopyCode := bInCopyCode, ParentObject := ParentObject);
END_METHOD

METHOD INTERNAL InvokeWithParams : ITcoTaskStatus
VAR_INPUT
    inDeceleration : UINT;
END_VAR
_deceleration    := inDeceleration;
InvokeWithParams := THIS^.Invoke();
END_METHOD

(*~
    <docu>
        <summary>
            Executes when task reaches the ```Done``` state .
        </summary>
    </docu>
~*)
METHOD PROTECTED OnDone
DriveRef.PlcToDrive.ControlSignal.STP := FALSE;
DriveRef.PlcToDrive.ControlSignal.RES := FALSE;
DriveRef.Restore();
END_METHOD

(*~
    <docu>
        <summary>
            Restores this instance to the Ready state. Can be called explicitly or from within one of the restore mechanisms.
            <para>
                See also <see cref="PlcDocu.TcoCore.TcoTask.AutoRestorable()"/>
            </para>
        </summary>
    </docu>
~*)
METHOD Restore : ITcoRestorable
SUPER^.Restore();
DriveRef.PlcToDrive.ControlSignal.STP := FALSE;
DriveRef.PlcToDrive.ControlSignal.RES := FALSE;
//DriveRef.Restore();
END_METHOD

END_FUNCTION_BLOCK
